(* IEC 61131-3 sources: repolevel_ST_code_completion/output/0127完整版本_带planner/repoeval_Command1/readful_result_before_fix, 12 files *)

(* ---- FB_AirConComfortCommand.st ---- *)
FUNCTION_BLOCK PUBLIC FB_AirConComfortCommand IMPLEMENTS I_Command
VAR
    targetTemperature : LREAL;
    targetFanSpeed    : INT;
    targetMode        : INT;
    bCommandExecuted  : BOOL;
END_VAR

VAR CONSTANT
    MODE_COOL : INT := 1;
    MODE_HEAT : INT := 2;
    MODE_FAN  : INT := 3;
END_VAR

VAR
    bIsOperable : BOOL;
END_VAR

// Initialize control parameters
targetTemperature := 22.0; // Default target temperature
targetFanSpeed := 2;       // Default fan speed
targetMode := MODE_COOL;   // Default mode

// Check if the air conditioning system is operable
IF __ISVALIDREF(refAirConditioning) THEN
    bIsOperable := refAirConditioning.bActive;
ELSE
    bIsOperable := FALSE;
END_IF

// Execute comfort command if operable
IF bIsOperable THEN
    refAirConditioning.SetTemperature(targetTemperature);
    refAirConditioning.SetFanSpeed(targetFanSpeed);
    CASE targetMode OF
        MODE_COOL: refAirConditioning.SetModeCool();
        MODE_HEAT: refAirConditioning.SetModeHeat();
        MODE_FAN:  refAirConditioning.SetModeFan();
    END_CASE;

    // Trigger hardware update
    refAirConditioning.Activate();
    bCommandExecuted := TRUE;
ELSE
    bCommandExecuted := FALSE;
END_IF

// Return execution result
RETURN;
END_FUNCTION_BLOCK

(* ---- FB_AirConditioning.st ---- *)
FUNCTION_BLOCK PUBLIC FB_AirConditioning
VAR_OUTPUT
	bActive			: BOOL;
	lrTemperature	: LREAL;
END_VAR
VAR
    lrDefaultTemperature : LREAL := 0.0;
    lrCalculatedTemperature : LREAL;
END_VAR

IF bActive THEN
    (* Calculate the current environment temperature based on control logic *)
    lrCalculatedTemperature := (* Insert temperature calculation logic here *);
    lrTemperature := lrCalculatedTemperature;
ELSE
    (* Set temperature to default value when inactive *)
    lrTemperature := lrDefaultTemperature;
END_IF;
END_FUNCTION_BLOCK

(* ---- FB_AirConStandbyCommand.st ---- *)
FUNCTION_BLOCK PUBLIC FB_AirConStandbyCommand IMPLEMENTS I_Command
VAR
    bStandbyCommandReceived : BOOL;
    bStandbyConditionsMet : BOOL;
    sExecutionResult : STRING;
END_VAR

bStandbyCommandReceived := FALSE;
bStandbyConditionsMet := FALSE;

// Step 1: Parse input command and check if it is "Standby"
IF __ISVALIDREF(refAirConditioning) THEN
    IF CommandType = "Standby" THEN
        bStandbyCommandReceived := TRUE;
    END_IF;
END_IF;

// Step 2: Check if the air conditioning system can enter standby mode
IF bStandbyCommandReceived THEN
    IF refAirConditioning.bActive AND (refAirConditioning.lrTemperature > 18.0 AND refAirConditioning.lrTemperature < 30.0) THEN
        bStandbyConditionsMet := TRUE;
    END_IF;
END_IF;

// Step 3: Execute standby operation if conditions are met
IF bStandbyConditionsMet THEN
    refAirConditioning.bActive := FALSE;
    sExecutionResult := 'Standby mode activated successfully';
ELSE
    sExecutionResult := 'Failed to activate standby mode';
END_IF;

// Step 4: Update internal system state or necessary flags
IF bStandbyConditionsMet THEN
    SystemState := 'Standby';
ELSE
    SystemState := 'Active';
END_IF;

// Step 5: Output execution result
ExecutionResult := sExecutionResult;
END_FUNCTION_BLOCK

(* ---- FB_CDPlayer.st ---- *)
FUNCTION_BLOCK PUBLIC FB_CDPlayer
VAR_OUTPUT
	bPlayerActive		: BOOL;
	byVolume			: BYTE;
	byTrack				: UINT;
END_VAR
VAR
	bCurrentState		: BOOL;
	byCurrentVolume		: BYTE;
	byCurrentTrack		: UINT;
END_VAR

bCurrentState := bPlayerActive;
byCurrentVolume := byVolume;
byCurrentTrack := byTrack;

IF bCurrentState THEN
	// Update outputs to reflect the current state of the CD player
	bPlayerActive := TRUE;
	byVolume := byCurrentVolume;
	byTrack := byCurrentTrack;
ELSE
	// If the player is not active, reset outputs
	bPlayerActive := FALSE;
	byVolume := 0;
	byTrack := 0;
END_IF;
END_FUNCTION_BLOCK

(* ---- FB_Lamp.st ---- *)
FUNCTION_BLOCK PUBLIC FB_Lamp
VAR_OUTPUT
	byLevel			: BYTE;
END_VAR
VAR
	byNewLevel		: BYTE;
END_VAR

IF byNewLevel < 0 THEN
	byLevel := 0;
ELSIF byNewLevel > 255 THEN
	byLevel := 255;
ELSE
	byLevel := byNewLevel;
END_IF;
END_FUNCTION_BLOCK

(* ---- FB_LampSetLevelCommand.st ---- *)
FUNCTION_BLOCK PUBLIC FB_LampSetLevelCommand IMPLEMENTS I_Command
VAR
	refLamp		: REFERENCE TO FB_Lamp;
	byNewLevel	: BYTE;
	bResult		: BOOL;
END_VAR

IF (__ISVALIDREF(refLamp)) THEN
	IF (byNewLevel > 100) THEN
		byNewLevel := 100; // Set to maximum allowed value if out of range
	ELSIF (byNewLevel < 0) THEN
		byNewLevel := 0; // Set to minimum allowed value if out of range
	END_IF

	bResult := refLamp.SetLevel(byNewLevel); // Update brightness level in hardware

	IF bResult THEN
		RETURN; // Command executed successfully
	END_IF
END_IF

bResult := FALSE; // Command execution failed
RETURN;
END_FUNCTION_BLOCK

(* ---- FB_MusicPlayCommand.st ---- *)
FUNCTION_BLOCK PUBLIC FB_MusicPlayCommand IMPLEMENTS I_Command
VAR
    isCommandActive : BOOL; // Indicates if the play command is active
    isPlaying : BOOL; // Indicates if music is currently playing
    errorStatus : BOOL; // Indicates if there was an error during execution
    logTimestamp : TIME; // Stores the timestamp of the last successful execution
END_VAR

IF NOT isCommandActive THEN
    RETURN;
END_IF;

IF __ISVALIDREF(refCDPlayer) THEN
    refCDPlayer.Start();
    IF refCDPlayer.IsPlaying THEN
        isPlaying := TRUE;
        errorStatus := FALSE;
        logTimestamp := TIME(); // Record the current timestamp
    ELSE
        isPlaying := FALSE;
        errorStatus := TRUE;
    END_IF;
ELSE
    errorStatus := TRUE;
END_IF;
END_FUNCTION_BLOCK

(* ---- FB_MusicStopCommand.st ---- *)
FUNCTION_BLOCK PUBLIC FB_MusicStopCommand IMPLEMENTS I_Command
VAR
    isCommandValid : BOOL;
    isStopSuccessful : BOOL;
END_VAR

IF __ISVALIDREF(THIS^.refCDPlayer) THEN
    isCommandValid := TRUE;
ELSE
    isCommandValid := FALSE;
END_IF;

IF isCommandValid THEN
    IF (THIS^.refCDPlayer.State = CDPlayerState.Playing) OR (THIS^.refCDPlayer.State = CDPlayerState.Paused) THEN
        THIS^.refCDPlayer.Stop();
        isStopSuccessful := (THIS^.refCDPlayer.State = CDPlayerState.Stopped);

        IF isStopSuccessful THEN
            // Update internal state to reflect the stop operation
            // (Assuming there is an internal state variable to update)
        ELSE
            // Handle stop failure
            // (Set error flag or status information as needed)
        END_IF;
    END_IF;
END_IF;
END_FUNCTION_BLOCK

(* ---- FB_Socket.st ---- *)
FUNCTION_BLOCK PUBLIC FB_Socket
VAR_OUTPUT
	bActive		: BOOL;
END_VAR
VAR
    bInitialized : BOOL := FALSE;
    bConnected   : BOOL := FALSE;
END_VAR

IF NOT bInitialized THEN
    (* Initialize the socket *)
    bInitialized := TRUE;
    bConnected := FALSE; (* Assume not connected initially *)
END_IF

(* Check the connection status *)
IF bInitialized THEN
    (* Simulate connection check logic *)
    IF bConnected THEN
        bActive := TRUE;
    ELSE
        bActive := FALSE;
    END_IF
END_IF

(* Update connection status for the next cycle *)
(* Simulate connection status change logic *)
bConnected := NOT bConnected; (* Toggle connection status for demonstration *)
END_FUNCTION_BLOCK

(* ---- FB_SocketOffCommand.st ---- *)
FUNCTION_BLOCK PUBLIC FB_SocketOffCommand IMPLEMENTS I_Command
VAR
    bCommandExecuted : BOOL := FALSE;
END_VAR

IF NOT bCommandExecuted THEN
    (* Step 1: Initialize command state *)
    bCommandExecuted := TRUE;

    (* Step 2: Call control logic to turn off the socket *)
    IF __ISVALIDREF(THIS^.refSocket) THEN
        THIS^.refSocket.Off();
    END_IF;

    (* Step 3: Update socket state to off *)
    IF __ISVALIDREF(THIS^.refSocket) THEN
        THIS^.refSocket.bActive := FALSE;
    END_IF;

    (* Step 4: Indicate command execution success *)
    bCommandExecuted := TRUE;
END_IF;

(* Step 5: Clean up resources if necessary *)
(* No additional resources to clean up in this implementation *)
END_FUNCTION_BLOCK

(* ---- FB_SocketOnCommand.st ---- *)
FUNCTION_BLOCK PUBLIC FB_SocketOnCommand IMPLEMENTS I_Command
VAR
    refSocket : REFERENCE TO FB_Socket;
    bCommandValid : BOOL;
END_VAR

VAR_INPUT
    sCommand : STRING;
END_VAR

VAR_OUTPUT
    bSuccess : BOOL;
    sErrorMessage : STRING;
END_VAR

VAR
    bSocketState : BOOL;
END_VAR

// Implementation
IF NOT __ISVALIDREF(refSocket) THEN
    bSuccess := FALSE;
    sErrorMessage := 'Invalid socket reference';
    RETURN;
END_IF

// Step 1: Initialize internal state variables
bCommandValid := FALSE;
bSocketState := FALSE;

// Step 2: Parse the command
IF sCommand = 'ON' THEN
    bCommandValid := TRUE;
    bSocketState := TRUE;
ELSIF sCommand = 'OFF' THEN
    bCommandValid := TRUE;
    bSocketState := FALSE;
ELSE
    bCommandValid := FALSE;
END_IF

// Step 3: Validate command parameters
IF NOT bCommandValid THEN
    bSuccess := FALSE;
    sErrorMessage := 'Invalid command';
    RETURN;
END_IF

// Step 4: Control the socket
IF bSocketState THEN
    refSocket.On();
ELSE
    refSocket.Off();
END_IF

// Step 5: Set output status
bSuccess := TRUE;
sErrorMessage := '';

// Step 6: Handle exceptions (already handled in validation steps above)
RETURN;
END_FUNCTION_BLOCK

(* ---- FB_SwitchPanel.st ---- *)
FUNCTION_BLOCK PUBLIC FB_SwitchPanel
VAR_INPUT
	arrSwitch		: ARRAY[1..8] OF BOOL;
END_VAR
VAR
	aiCommand		: ARRAY[1..8] OF I_Command;
	arrRtrig		: ARRAY[1..8] OF R_TRIG;
	nIndex			: INT;
END_VAR

FOR nIndex := 1 TO 8 DO
	arrRtrig[nIndex](CLK := arrSwitch[nIndex]);
	IF arrRtrig[nIndex].Q THEN
		IF (aiCommand[nIndex] <> 0) THEN
			aiCommand[nIndex].Execute();
		END_IF
	END_IF
END_FOR
END_FUNCTION_BLOCK
